FUNCTION_BLOCK FB_Count
VAR_INPUT
	bCount 			: BOOL;
	nCountIncrement : INT := 1;
END_VAR
VAR_OUTPUT
	nCounterValue : INT;
END_VAR
VAR
	rtCount : R_TRIG;
END_VAR

rtCount(CLK := bCount);
IF rtCount.Q THEN
	nCounterValue := nCounterValue + nCountIncrement;
END_IF

END_FUNCTION_BLOCK

(* stored: Version 1.1.0.1, ProductVersion 3.1.4024.12
   POU FB_Count: Id {843bd016-1464-46f3-b6f9-76f43cb76bf9}, SpecialFunc None *)
